{attribute 'qualified_only'}
{attribute 'strict'}
{attribute 'to_string'}
TYPE E_PhaseSelect :
(
	ALL := 0,
    L1,
    L2,
    L3
);
END_TYPE

(* stored: Version 1.1.0.1
   DUT E_PhaseSelect: Id {33075ffc-ab43-4ae0-88ee-68b6798ae8e1} *)
